TYPE "MEStoPLC_AGVExchange"
VERSION : 0.1
   STRUCT
      "M-PosCallDone1" : Byte;
      "M-PosCallDone2" : Byte;
      "M-PosCallDone3" : Byte;
      "M-PosCallDone4" : Byte;
      "M-PosCallDone5" : Byte;
      Reserve : Array[1..994] of Byte;
   END_STRUCT;

END_TYPE

